FUNCTION_BLOCK MachineContainer EXTENDS ZCore.ObjectContainer
VAR_INPUT
END_VAR
VAR_OUTPUT
END_VAR
VAR
  {attribute 'hide'}
  _parent : REFERENCE TO MachineUnit;
END_VAR

{attribute 'hide' }
METHOD FB_init : BOOL
VAR_INPUT
	bInitRetains : BOOL; // if TRUE, the retain variables are initialized (warm start / cold start)
	bInCopyCode : BOOL;  // if TRUE, the instance afterwards gets moved into the copy code (online change)
  unit : REFERENCE TO MachineUnit;
END_VAR
_parent REF= unit;
END_METHOD

END_FUNCTION_BLOCK

(* stored: Version 1.1.0.1
   POU MachineContainer: Id {7c87ade7-958c-4a2e-8fac-b91119cc3a37}, SpecialFunc None
   Method FB_init: Id {cc27ab95-0061-4949-be44-313051e27d52} *)
